FUNCTION_BLOCK AX_ASR_SWITCH (* Converts AX adapter to ASR adapter (1:1 mapping: TRUE=SET, FALSE=RESET) *)
  (* Standard: 61499-2; Description: Copyright (c) 2026 HR Agrartechnik GmbH This program and the accompanying materials are made available under the terms of the Eclipse Public License 2.0 which is available at https://www.eclipse.org/legal/epl-2.0/ SPDX-License-Identifier: EPL-2.0 *)
  (* Version 1.0, 2026-01-17, Franz Höpfinger, HR Agrartechnik GmbH *)
  PACKAGE adapter::events::unidirectional;
  IMPORT iec61499::events::E_SWITCH;
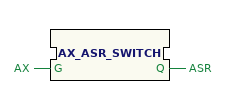
  SOCKETS
    G : adapter::types::unidirectional::AX; (* Boolean Input *)
  END_SOCKETS
  PLUGS
    Q : adapter::types::unidirectional::ASR; (* Set/Reset Output *)
  END_PLUGS
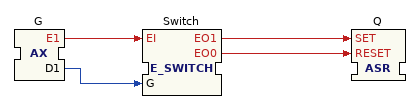
  FBS
    Switch : iec61499::events::E_SWITCH;
  END_FBS
  EVENT_CONNECTIONS
    G.E1 TO Switch.EI;
    Switch.EO1 TO Q.SET;
    Switch.EO0 TO Q.RESET;
  END_CONNECTIONS
  DATA_CONNECTIONS
    G.D1 TO Switch.G;
  END_CONNECTIONS
END_FUNCTION_BLOCK
